INTERFACE IStation

PROPERTY Enabled : BOOL
GET
END_GET
SET
END_SET
END_PROPERTY

METHOD Execute
VAR_INPUT
END_VAR
END_METHOD

PROPERTY Index : DINT
GET
END_GET
SET
END_SET
END_PROPERTY

END_INTERFACE

(* stored: Version 1.1.0.1
   Itf IStation: Id {ff1f012a-557f-4092-a110-cbfea7b12f66}
   Property Enabled: Id {bcdec233-c136-4ced-a9f3-6409b2f70365}
   Get Get: Id {2a0a2e04-2229-439a-a1dd-06fa563021d5}
   Set Set: Id {a35044b9-82c5-4ae0-9020-63e66ad1e291}
   Method Execute: Id {1c99f3c0-b0d7-4a9a-8630-8b442b94cb12}
   Property Index: Id {a79859f1-b9e2-4a24-92e1-6121500e96bd}
   Get Get: Id {36f288f1-c4d9-4fb9-bdb7-96f51fe63f0e}
   Set Set: Id {6b03bcb8-136f-4359-b2bb-5674f0aa092d} *)
